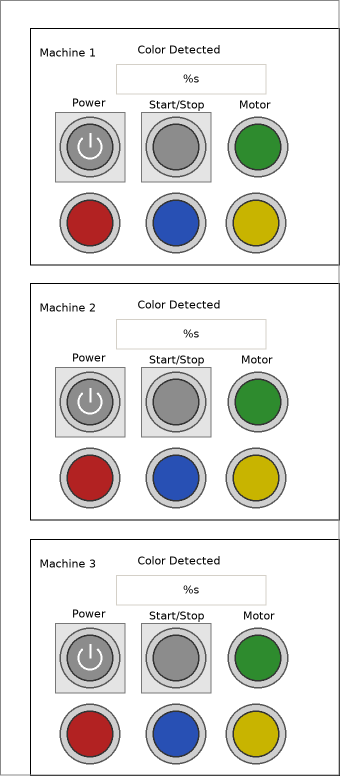
VISUALIZATION Visualization  // 340x776
    Rectangle (30,28 310x237)
    Lamp1 (223,112 70x70), variable: MAIN.machine1.conveyor.bRunning, style: Lamp-Lamp1-Green
    Label (30,29 76x48), "Machine 1"
    Textfield (116,64 150x30), "%s", text variable: MAIN.machine1.currentColor
    Lamp1 (55,188 70x70), variable: MAIN.machine1.redDiverter.bActive, style: Lamp-Lamp1-Red
    Lamp1 (141,188 70x70), variable: MAIN.machine1.blueDiverter.bActive, style: Lamp-Lamp1-Blue
    Lamp1 (221,188 70x70), variable: MAIN.machine1.yellowDiverter.bActive, style: Lamp-Lamp1-Yellow
    Label (102,21 154x58), "Color Detected"
    PushSwitch (141,112 70x70), variable: MAIN.machine1.conveyor.bRunning, behaviour: TOGGLE, style: Switch-PushSwitch-Gray
    PowerSwitch (55,112 70x70), variable: MAIN.machine1.bEnabled, behaviour: TOGGLE, style: Switch-PowerSwitch-Gray
    Label (53,87 72x32), "Power"
    Label (141,89 72x32), "Start/Stop"
    Rectangle (30,283 310x237)
    Lamp1 (223,367 70x70), variable: MAIN.machine2.conveyor.bRunning, style: Lamp-Lamp1-Green
    Label (30,284 76x48), "Machine 2"
    Textfield (116,319 150x30), "%s", text variable: MAIN.machine2.currentColor
    Lamp1 (55,443 70x70), variable: MAIN.machine2.redDiverter.bActive, style: Lamp-Lamp1-Red
    Lamp1 (141,443 70x70), variable: MAIN.machine2.blueDiverter.bActive, style: Lamp-Lamp1-Blue
    Lamp1 (221,443 70x70), variable: MAIN.machine2.yellowDiverter.bActive, style: Lamp-Lamp1-Yellow
    Label (102,276 154x58), "Color Detected"
    PushSwitch (141,367 70x70), variable: MAIN.machine2.conveyor.bRunning, behaviour: TOGGLE, style: Switch-PushSwitch-Gray
    PowerSwitch (55,367 70x70), variable: MAIN.machine2.bEnabled, behaviour: TOGGLE, style: Switch-PowerSwitch-Gray
    Label (53,342 72x32), "Power"
    Label (141,344 72x32), "Start/Stop"
    Rectangle (30,539 310x237)
    Lamp1 (223,623 70x70), variable: MAIN.machine3.conveyor.bRunning, style: Lamp-Lamp1-Green
    Label (30,540 76x48), "Machine 3"
    Textfield (116,575 150x30), "%s", text variable: MAIN.machine3.currentColor
    Lamp1 (55,699 70x70), variable: MAIN.machine3.redDiverter.bActive, style: Lamp-Lamp1-Red
    Lamp1 (141,699 70x70), variable: MAIN.machine3.blueDiverter.bActive, style: Lamp-Lamp1-Blue
    Lamp1 (221,699 70x70), variable: MAIN.machine3.yellowDiverter.bActive, style: Lamp-Lamp1-Yellow
    Label (102,532 154x58), "Color Detected"
    PushSwitch (141,623 70x70), variable: MAIN.machine3.conveyor.bRunning, behaviour: TOGGLE, style: Switch-PushSwitch-Gray
    PowerSwitch (55,623 70x70), variable: MAIN.machine3.bEnabled, behaviour: TOGGLE, style: Switch-PowerSwitch-Gray
    Label (53,598 72x32), "Power"
    Label (141,600 72x32), "Start/Stop"
    Label (221,344 72x32), "Motor"
    Label (219,89 72x32), "Motor"
    Label (223,600 72x32), "Motor"
END_VISUALIZATION

(* stored: Version 1.1.0.1
   Visu Visualization: Id {537b8653-28d0-414a-a917-0dad71d7675b} *)
